FUNCTION_BLOCK FB_File
VAR
    eMode: 					SysFile.ACCESS_MODE := SysFile.AM_APPEND_PLUS;
    hFile: 					SysFile.SysTypes.RTS_IEC_HANDLE;
	Result:					SysFile.SysTypes.RTS_IEC_RESULT;
	pResult:				POINTER TO SysFile.SysTypes.RTS_IEC_RESULT:= ADR(Result);
    pBuffer:				POINTER TO BYTE;
    nBuffer:				UDINT;
END_VAR

// Closes the currently opened file.
METHOD PUBLIC M_Close : BOOL
VAR_INPUT
END_VAR
IF hFile <> SysFile.SysTypes.RTS_INVALID_HANDLE THEN
   pResult^:= SysFile.SysFileClose(hFile);
END_IF

M_Close:= TRUE;
END_METHOD

// Delete file
METHOD PUBLIC M_Delete : BOOL
VAR_INPUT
    sFileName : STRING(255);
END_VAR
pResult^:= SysFile.SysFileDelete(sFileName);
M_Delete:= TRUE;
END_METHOD

METHOD PUBLIC M_GetSize : UDINT
VAR_INPUT
END_VAR
M_GetSize:= LWORD_TO_UDINT(SysFile.SysFileGetSizeByHandle(hFile, pResult));
END_METHOD

// Open file
METHOD PUBLIC M_Open : BOOL
VAR_INPUT
    sFileName:				STRING(255);
END_VAR
hFile := SysFile.SysFileOpen(sFileName, eMode, pResult);

M_Open := true;
END_METHOD

// Read file
METHOD PUBLIC M_Read : BOOL
VAR_INPUT
END_VAR
IF pBuffer <> 0 THEN
	__DELETE(pBuffer);
	nBuffer:= 0;
END_IF

nBuffer:= M_GetSize();
pBuffer:= __NEW(BYTE, nBuffer);
SysFile.SysFileRead(hFile, pBuffer, nBuffer, pResult );

M_Read := TRUE;
END_METHOD

METHOD PUBLIC M_Size : UDINT
VAR_INPUT
END_VAR
SysFile.SysFileGetSizeByHandle(hFile, pResult);
END_METHOD

// Closes the currently opened file.
METHOD PUBLIC M_Status : BOOL
VAR_INPUT
END_VAR
IF hFile <> SysFile.SysTypes.RTS_INVALID_HANDLE THEN
   pResult^:= SysFile.SysFileGetStatus(hFile);
END_IF

M_Close:= TRUE;
END_METHOD

// Writes the contents of the buffer into a file.
METHOD PUBLIC M_Write : BOOL
VAR_INPUT
	sValue:			STRING(255);
END_VAR
IF hFile <> SysFile.SysTypes.RTS_INVALID_HANDLE THEN
    SysFile.SysFileWrite(hFile := hFile,
                         pbyBuffer := ADR(sValue),
                         ulSize := len(sValue),
                         pResult := pResult);
END_IF

M_Write:= TRUE;
END_METHOD

END_FUNCTION_BLOCK

(* stored: Version 1.1.0.1
   POU FB_File: Id {879562f4-6da1-45fb-a1f3-48bd69fd0a1e}, SpecialFunc None
   Method M_Close: Id {2032b7d9-4eba-4de7-bc38-d769b85ee782}
   Method M_Delete: Id {031610a1-66f5-45ab-8b86-edea27263a7f}
   Method M_GetSize: Id {da2b00f7-d9aa-4c86-85c6-4fdbc9147466}
   Method M_Open: Id {6307849d-083a-4a2a-8a54-cacfa983025c}
   Method M_Read: Id {4210ba0d-c339-4c83-b89a-8d5ea8fd601c}
   Method M_Size: Id {3fcaa98d-265e-4de4-91e2-fd9b15df9b65}
   Method M_Status: Id {8f0ab01f-d98a-40bc-9f73-79c89b4ed20b}
   Method M_Write: Id {b956b515-594f-440e-be50-f979325c8ffe} *)
